# EPICS substitutions: ioc/SRS300App/Db/devSRS_PS375.substitutions
##########################################################################
# Copyright (c) 2012 Lawrence Berkeley National Laboratory, Accelerator
# Technology Group, Engineering Division
# This code is distributed subject to a Software License Agreement found
# in file LICENSE that is included with this distribution.
##########################################################################

file "$(TOP)/db/devSRS_PS3xx.template"
{
  #VMIN = Minimum voltage and minimum step size, VMAX = maximum voltage
  #IMIN and IMAX = Minimum and maximum current, respectively
  #POLARITY = Polarity of the device (for now, 0=positive)
  #TOLERANCE = Voltage amount the device may be inaccurate by at higher voltage levels.
  #PREC = decimal point accuracy of values
  { VMIN="100", VMAX="20000", IMIN="0", IMAX="525e-6", POLARITY="0", TOLERANCE="4", PREC = "2" }
}
